SUBAPPLICATION Uebung_001c3_AX (* DigitalInput_I1 auf DigitalOutput_Q1 --> Eingang abfragen bei Boot. *)
  (* Standard: 61499-2; Description: Copyright (c) 2026 Meisterschulen am Ostbahnhof This program and the accompanying materials are made available under the terms of the Eclipse Public License 2.0 which is available at https://www.eclipse.org/legal/epl-2.0/ SPDX-License-Identifier: EPL-2.0 *)
  (* Version 1.0, 2026-09-09, Franz Höpfinger, Meisterschulen am Ostbahnhof, initial API and implementation and/or initial documentation *)
  PACKAGE Uebungen;
  IMPORT logiBUS::io::DI::logiBUS_DI::Input_I1;
  IMPORT logiBUS::io::DQ::logiBUS_DO::Output_Q1;
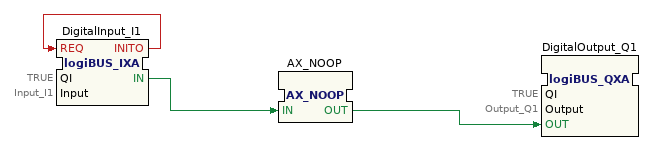
  (* ohne die Linie INITO->REQ ist der Ausgang Q1 beim Start FALSE. mit der Linie ist er TRUE. *)
  (* In Adapter-Architektur entspricht der doppelten Negierung (NOT an NOT) der Baustein AX_NOOP. *)
  FBS
    DigitalOutput_Q1 : logiBUS::io::DQ::logiBUS_QXA(QI := TRUE, Output := Output_Q1);
    DigitalInput_I1 : logiBUS::io::DI::logiBUS_IXA(QI := TRUE, Input := Input_I1);
    AX_NOOP : adapter::booleanOperators::AX_NOOP;
  END_FBS
  EVENT_CONNECTIONS
    DigitalInput_I1.INITO TO DigitalInput_I1.REQ;
  END_CONNECTIONS
  ADAPTER_CONNECTIONS
    DigitalInput_I1.IN TO AX_NOOP.IN;
    AX_NOOP.OUT TO DigitalOutput_Q1.OUT;
  END_CONNECTIONS
END_SUBAPPLICATION
